// LS Electric XG5000 project: 과년70_3_수정
// PLC NewPLC
// module base 0 slot 0: 입출력 모듈:XBC-DR20S (DC 24V 입력 12점, 릴레이 출력 8점)

PROGRAM NewProgram (task: 스캔 프로그램)

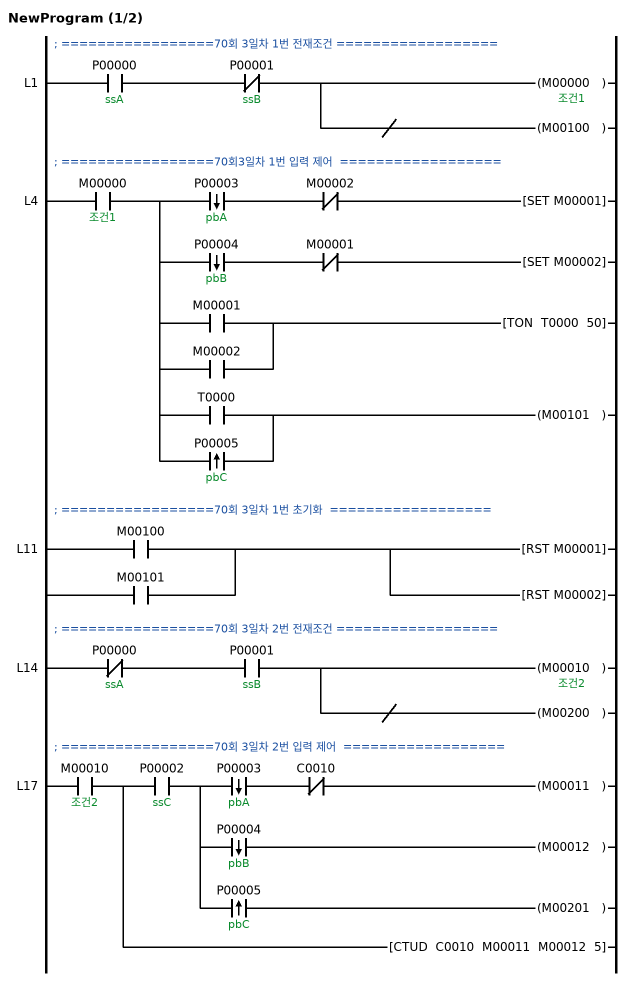
// =================70회 3일차 1번 전재조건 ==================
; L1
LOAD      P00000	// ssA
AND NOT   P00001	// ssB
OUT       M00000	// 조건1
NOT
OUT       M00100
// =================70회3일차 1번 입력 제어  ==================
; L4
LOAD      M00000	// 조건1
MPUSH
ANDN      P00003	// pbA
AND NOT   M00002
SET       M00001
MLOAD
ANDN      P00004	// pbB
AND NOT   M00001
SET       M00002
MLOAD
LOAD      M00001
OR        M00002
AND LOAD
TON       T0000 50
MPOP
LOAD      T0000
ORP       P00005	// pbC
AND LOAD
OUT       M00101
// =================70회 3일차 1번 초기화  ==================
; L11
LOAD      M00100
OR        M00101
RST       M00001
RST       M00002
// =================70회 3일차 2번 전재조건 ==================
; L14
LOAD NOT  P00000	// ssA
AND       P00001	// ssB
OUT       M00010	// 조건2
NOT
OUT       M00200
// =================70회 3일차 2번 입력 제어  ==================
; L17
LOAD      M00010	// 조건2
MPUSH
AND       P00002	// ssC
MPUSH
ANDN      P00003	// pbA
AND NOT   C0010
OUT       M00011
MLOAD
ANDN      P00004	// pbB
OUT       M00012
MPOP
ANDP      P00005	// pbC
OUT       M00201
MPOP
CTUD      C0010 M00011 M00012 5

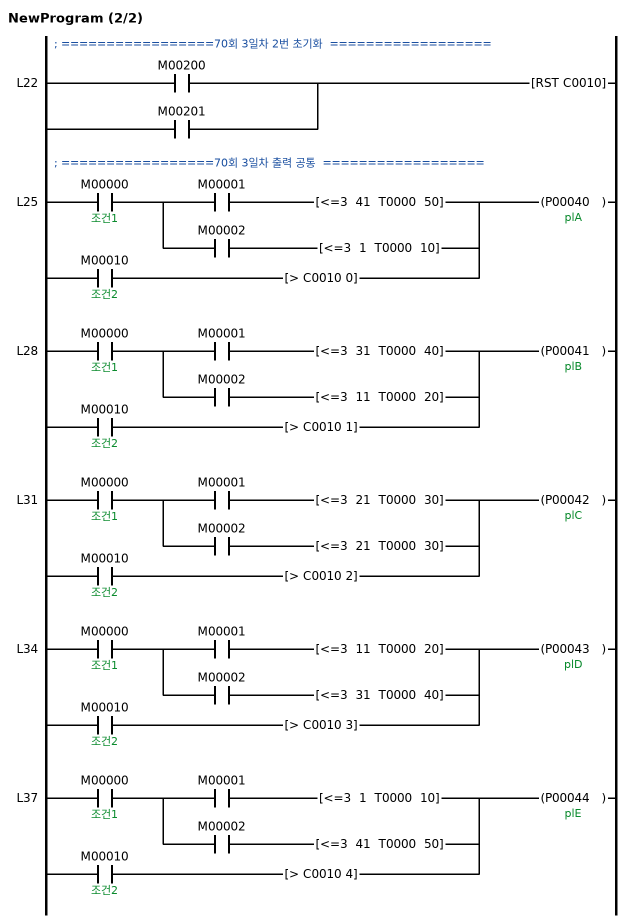
// =================70회 3일차 2번 초기화  ==================
; L22
LOAD      M00200
OR        M00201
RST       C0010
// =================70회 3일차 출력 공통  ==================
; L25
LOAD      M00000	// 조건1
LOAD      M00001
AND<=3    41 T0000 50
LOAD      M00002
AND<=3    1 T0000 10
OR LOAD
AND LOAD
LOAD      M00010	// 조건2
AND>      C0010 0
OR LOAD
OUT       P00040	// plA
; L28
LOAD      M00000	// 조건1
LOAD      M00001
AND<=3    31 T0000 40
LOAD      M00002
AND<=3    11 T0000 20
OR LOAD
AND LOAD
LOAD      M00010	// 조건2
AND>      C0010 1
OR LOAD
OUT       P00041	// plB
; L31
LOAD      M00000	// 조건1
LOAD      M00001
AND<=3    21 T0000 30
LOAD      M00002
AND<=3    21 T0000 30
OR LOAD
AND LOAD
LOAD      M00010	// 조건2
AND>      C0010 2
OR LOAD
OUT       P00042	// plC
; L34
LOAD      M00000	// 조건1
LOAD      M00001
AND<=3    11 T0000 20
LOAD      M00002
AND<=3    31 T0000 40
OR LOAD
AND LOAD
LOAD      M00010	// 조건2
AND>      C0010 3
OR LOAD
OUT       P00043	// plD
; L37
LOAD      M00000	// 조건1
LOAD      M00001
AND<=3    1 T0000 10
LOAD      M00002
AND<=3    41 T0000 50
OR LOAD
AND LOAD
LOAD      M00010	// 조건2
AND>      C0010 4
OR LOAD
OUT       P00044	// plE